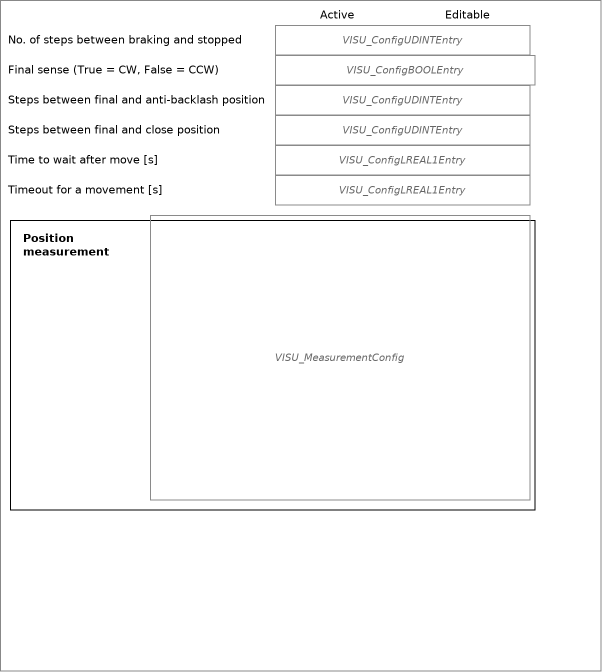
VISUALIZATION VISU_M2Config_AxisGeneral  // 602x672
VAR_IN_OUT
    editable : M2AxisGeneralConfig;
	active : M2AxisGeneralConfig;
END_VAR
    Label (275,5 125x20), "Active"
    Label (405,5 125x20), "Editable"
    Label (5,25 250x30), "No. of steps between braking and stopped"
    Frame (275,25 255x30), tooltip "The number of steps to be expected between the time at which the PLC realizes that the brake signal must be set, and the time that the axis is fully stopped (for Z axis: at low speed)"
        shows VISU_ConfigUDINTEntry(active := active.stoppingSteps, editable := editable.stoppingSteps)
    Label (5,55 285x30), "Final sense (True = CW, False = CCW)"
    Label (5,85 285x30), "Steps between final and anti-backlash position"
    Frame (275,55 260x30), tooltip "The number of steps which should be carried out at minimum to counter-act the backlash in the system during the final move (for Z axis: at low speed)"
        shows VISU_ConfigBOOLEntry(active := active.finalSenseCW, editable := editable.finalSenseCW)
    Frame (275,85 255x30), tooltip "The number of steps which should be carried out at minimum to counter-act the backlash in the system during the final move (for Z axis: at low speed)"
        shows VISU_ConfigUDINTEntry(active := active.antiBacklashPosition, editable := editable.antiBacklashPosition)
    Frame (275,115 255x30), tooltip "The number of steps which should be carried out at minimum to counter-act the backlash in the system during the final move (for Z axis: at low speed)"
        shows VISU_ConfigUDINTEntry(active := active.closePosition, editable := editable.closePosition)
    Label (5,115 265x30), "Steps between final and close position"
    Rectangle (10,220 525x290)
    Label (5,145 285x30), "Time to wait after move [s]"
    Frame (275,145 255x30), tooltip "Time (in seconds) to wait after the axis has been moved"
        shows VISU_ConfigLREAL1Entry(active := active.waitAfterMove, editable := editable.waitAfterMove)
    Frame (275,175 255x30), tooltip "Time (in seconds) to wait after the axis has been moved"
        shows VISU_ConfigLREAL1Entry(active := active.timeout, editable := editable.timeout)
    Label (5,175 285x30), "Timeout for a movement [s]"
    Frame (150,215 380x285)
        shows VISU_MeasurementConfig(active := active.measurement, editable := editable.measurement)
    Label (20,230 150x30), "Position measurement"
    Line (600,670)
END_VISUALIZATION

(* stored: Version 1.1.0.1, ProductVersion 3.1.4019.2
   Visu VISU_M2Config_AxisGeneral: Id {fb7e073e-7bb9-4170-af81-2e45d4416bd8} *)
